FUNCTION_BLOCK Axis EXTENDS CyclicComponent IMPLEMENTS I_Initializable, I_Axis
VAR
	_Axis				 : REFERENCE TO AXIS_REF;
	Defaults			 : ST_MotionDefaults;
	MotionTaskCollection : MotionTaskCollection<ApplicationBaseMotionParameterNc2.MaxMotionTasks>(THIS^);

	// Tasks
	{attribute 'hide'}
	PowerTask : PowerTask := (Name := 'MC Power');
	{attribute 'hide'}
	JogTask : MoveJogTask := (Name := 'MC Jog');
	{attribute 'hide'}
	_StopTask : I_MotionTask := Defaults.DefaultStopTask;
	{attribute 'hide'}
	_ResetTask : I_MotionTask := Defaults.DefaultResetTask;
	{attribute 'hide'}
	_HomeTask : I_MotionTask := Defaults.DefaultHomeTask;

	//
	{attribute 'hide'}
	MCReadParameterSet : MC_ReadParameterSet;
	_AxisParameters	   : ST_AxisParameterSet;
	{attribute 'hide'}
	_Initialized : BOOL;
	{attribute 'hide'}
	_Acceleration : LREAL;
	{attribute 'hide'}
	_Deceleration : LREAL;
	{attribute 'hide'}
	_Velocity : LREAL;
	{attribute 'hide'}
	_Jerk		  : LREAL;
	_McBufferMode : MC_BufferMode;
	_MoveOptions  : ST_MoveOptions;
END_VAR

{attribute 'monitoring' := 'call'}
PROPERTY Acceleration : LREAL
GET
Acceleration := _Acceleration;
END_GET
SET
_Acceleration := Acceleration;
END_SET
END_PROPERTY

{attribute 'monitoring' := 'call'}
PROPERTY ActualAcceleration : LREAL
GET
ActualAcceleration := _Axis.NcToPlc.ActAcc;
END_GET
END_PROPERTY

{attribute 'monitoring' := 'call'}
PROPERTY ActualPosition : LREAL
GET
ActualPosition := _Axis.NcToPlc.ActPos;
END_GET
END_PROPERTY

{attribute 'monitoring' := 'call'}
PROPERTY ActualPositionModulo : LREAL
GET
ActualPositionModulo := _Axis.NcToPlc.ModuloActPos;
END_GET
END_PROPERTY

{attribute 'monitoring' := 'call'}
PROPERTY ActualTorque : LREAL
GET
ActualTorque := _Axis.NcToPlc.ActTorque;
END_GET
END_PROPERTY

{attribute 'monitoring' := 'call'}
PROPERTY ActualVelocity : LREAL
GET
ActualVelocity := _Axis.NcToPlc.ActVelo;
END_GET
END_PROPERTY

PROPERTY Axis : REFERENCE TO AXIS_REF
GET
Axis REF= _Axis;
END_GET
END_PROPERTY

PROPERTY AxisParameterSet : REFERENCE TO ST_AxisParameterSet
GET
AxisParameterSet REF= _AxisParameters;
END_GET
END_PROPERTY

PROPERTY BufferMode : REFERENCE TO MC_BufferMode
GET
BufferMode REF= _McBufferMode;
END_GET
END_PROPERTY

{attribute 'monitoring' := 'call'}
PROPERTY Busy : BOOL
GET
Busy := MotionTaskCollection.Busy;
END_GET
END_PROPERTY

METHOD CyclicLogic
IF NOT _Initialized THEN
	Initialize();
	RETURN;
END_IF

_Axis.ReadStatus();
MotionTaskCollection.CyclicLogic();
END_METHOD

{attribute 'monitoring' := 'call'}
PROPERTY Deceleration : LREAL
GET
Deceleration := _Deceleration;
END_GET
SET
_Deceleration := Deceleration;
END_SET
END_PROPERTY

METHOD Disable
PowerTask.Disable();
END_METHOD

METHOD Enable
IF Error THEN
	RETURN;
END_IF

PowerTask.Enable();
END_METHOD

{attribute 'monitoring' := 'call'}
PROPERTY Enabled : BOOL
GET
Enabled := PowerTask.Enabled;
END_GET
END_PROPERTY

{attribute 'monitoring' := 'call'}
PROPERTY Error : BOOL
GET
Error := MotionTaskCollection.Error OR _Axis.Status.Error;
END_GET
END_PROPERTY

{attribute 'monitoring' := 'call'}
PROPERTY ErrorId : UDINT
GET
IF _Axis.Status.ErrorID <> 0 THEN
	ErrorId := _Axis.Status.ErrorID;
	RETURN;
END_IF

ErrorId := MotionTaskCollection.ErrorId;
END_GET
END_PROPERTY

(*FB_Init is always available implicitly and it is used primarily for initialization.
The return value is not evaluated. For a specific influence, you can also declare the
methods explicitly and provide additional code there with the standard initialization
code. You can evaluate the return value.*)
METHOD FB_Init : BOOL
VAR_INPUT
	(* TRUE: the retain variables are initialized (reset warm / reset cold)*)
	bInitRetains : BOOL;

	(* TRUE: the instance will be copied to the copy code afterward (online change)   *)
	bInCopyCode : BOOL;
	Name		: T_MaxString;
	Axis		: REFERENCE TO AXIS_REF;
END_VAR
_Axis REF= Axis;

// Register all Motion Tasks to Collection
MotionTaskCollection.AddTask(PowerTask);
MotionTaskCollection.AddTask(_StopTask);
MotionTaskCollection.AddTask(_ResetTask);
MotionTaskCollection.AddTask(_HomeTask);
MotionTaskCollection.AddTask(JogTask);
END_METHOD

METHOD Home
VAR_INPUT
END_VAR
_HomeTask.Execute();
END_METHOD

PROPERTY HomeTask : I_MotionTask
SET
MotionTaskCollection.RemoveTaskByInstance(_HomeTask);
_HomeTask := HomeTask;
MotionTaskCollection.AddTask(_HomeTask);
END_SET
END_PROPERTY

{attribute 'monitoring' := 'call'}
PROPERTY InhibitFeedBackward : BOOL
GET
InhibitFeedBackward := PowerTask.InhibitFeedBackward;
END_GET
SET
PowerTask.InhibitFeedBackward := InhibitFeedBackward;
END_SET
END_PROPERTY

{attribute 'monitoring' := 'call'}
PROPERTY InhibitFeedForward : BOOL
GET
InhibitFeedForward := PowerTask.InhibitFeedForward;
END_GET
SET
PowerTask.InhibitFeedForward := InhibitFeedForward;
END_SET
END_PROPERTY

METHOD Initialize
IF NOT _Initialized THEN
	MCReadParameterSet(Parameter := _AxisParameters, Axis := _Axis, Execute := TRUE);
	IF NOT MCReadParameterSet.Busy THEN
		IF MCReadParameterSet.Error THEN
			Trace.LogMessage(_Name, 'Axis not initialized - McReadParameter failed!');
		ELSIF MCReadParameterSet.Done THEN
			_Velocity	  := _AxisParameters.fVeloSlowManual;
			_Acceleration := _AxisParameters.fAcceleration;
			_Deceleration := _AxisParameters.fDeceleration;
			_Jerk		  := _AxisParameters.fJerk;
			Trace.LogMessage(_Name, 'Axis initialization complete');
			_Initialized := TRUE;
		END_IF

		MCReadParameterSet(Parameter := _AxisParameters, Axis := _Axis, Execute := FALSE);
	END_IF
END_IF
END_METHOD

{attribute 'monitoring' := 'call'}
PROPERTY Initialized : BOOL
GET
Initialized := _Initialized;
END_GET
SET
_Initialized := Initialized;
END_SET
END_PROPERTY

{attribute 'monitoring' := 'call'}
PROPERTY Jerk : LREAL
GET
Jerk := _Jerk;
END_GET
SET
_Jerk := Jerk;
END_SET
END_PROPERTY

METHOD Jog
VAR_INPUT
	JogForward	 : BOOL;
	JogBackwards : BOOL;
	JogMode		 : E_JogMode := E_JogMode.MC_JOGMODE_STANDARD_SLOW;
	Position	 : LREAL	 := 0;
END_VAR
IF Error THEN
	RETURN;
END_IF

JogTask.JogBackwards := JogBackwards;
JogTask.JogForward	 := JogForward;
JogTask.Position	 := Position;
JogTask.Mode		 := JogMode;
JogTask.Execute();
END_METHOD

PROPERTY MotionTasks : I_MotionTaskCollection
GET
MotionTasks := MotionTaskCollection;
END_GET
END_PROPERTY

PROPERTY MoveOptions : REFERENCE TO ST_MoveOptions
GET
MoveOptions REF= _MoveOptions;
END_GET
END_PROPERTY

{attribute 'monitoring' := 'call'}
PROPERTY Override : LREAL
SET
PowerTask.Override := Override;
END_SET
END_PROPERTY

{attribute 'monitoring' := 'call'}
PROPERTY PositionLag : LREAL
GET
PositionLag := _Axis.NcToPlc.PosDiff;
END_GET
END_PROPERTY

METHOD RegisterWithParent
VAR_INPUT
	Parent : I_ContainComponents;
END_VAR
SUPER^.RegisterWithParent(Parent);
Parent.RegisterInitialize(THIS^);
END_METHOD

METHOD Reset
IF _ResetTask.Execute() THEN
	MotionTaskCollection.Reset();
END_IF
END_METHOD

PROPERTY ResetTask : I_MotionTask
SET
MotionTaskCollection.RemoveTaskByInstance(_ResetTask);
_ResetTask := ResetTask;
MotionTaskCollection.AddTask(_ResetTask);
END_SET
END_PROPERTY

{attribute 'monitoring' := 'call'}
PROPERTY SetAcceleration : LREAL
GET
SetAcceleration := _Axis.NcToPlc.SetAcc;
END_GET
END_PROPERTY

{attribute 'monitoring' := 'call'}
PROPERTY SetPosition : LREAL
GET
SetPosition := _Axis.NcToPlc.SetPos;
END_GET
END_PROPERTY

{attribute 'monitoring' := 'call'}
PROPERTY SetPositionModulo : LREAL
GET
SetPositionModulo := _Axis.NcToPlc.ModuloSetPos;
END_GET
END_PROPERTY

{attribute 'monitoring' := 'call'}
PROPERTY SetVelocity : LREAL
GET
SetVelocity := _Axis.NcToPlc.SetVelo;
END_GET
END_PROPERTY

METHOD Stop
IF Error AND _Axis.Status.Error THEN
	(* It's possible that a function block errored but
	not the NC itself--in this case we can allow a stop command.
	If the NC Axis has a real fault then we want a successful reset first *)
	RETURN;
END_IF

_StopTask.Execute();
END_METHOD

{attribute 'monitoring' := 'call'}
PROPERTY Stopped : BOOL
GET
Stopped := _Axis.Status.NotMoving;
END_GET
END_PROPERTY

PROPERTY StopTask : I_MotionTask
SET
MotionTaskCollection.RemoveTaskByInstance(_StopTask);
_StopTask := StopTask;
MotionTaskCollection.AddTask(_ResetTask);
END_SET
END_PROPERTY

{attribute 'monitoring' := 'call'}
PROPERTY Velocity : LREAL
GET
Velocity := _Velocity;
END_GET
SET
_Velocity := Velocity;
END_SET
END_PROPERTY

END_FUNCTION_BLOCK

(* stored: Version 1.1.0.1, ProductVersion 3.1.4026.18
   POU Axis: Id {c3c03e8a-759c-4ce9-bcae-63318d943e7c}, SpecialFunc None
   Folder Component: Id {b9674294-e5e8-4857-b2dd-bb9605b4f949}
   Folder Cyclic: Id {cd62d491-a87a-4c24-ab53-621ad021711e}
   Folder Dynamics: Id {393c3e99-a69d-4243-96b4-7490d06ba075}
   Folder Enable: Id {a996dd7a-39c8-423c-9839-645e36a4c7ae}
   Folder Home: Id {e215008b-3961-4321-9331-07c098f36434}
   Folder Initialize: Id {350a9f43-6c08-4c9b-bd16-bb4fcd640dda}
   Folder Jog: Id {b440d357-8c50-41b7-97b2-91a6c011f5d6}
   Folder Reset: Id {853c8cf9-dc4d-4635-94bf-40639ab6791d}
   Folder Status: Id {72a29854-77b1-4e21-8c83-e6fb17183b47}
   Folder Stop: Id {4b02773b-6d51-4517-a15d-46b46992d36e}
   Property Acceleration: Id {bc2c3c5d-a4a9-4cb5-98d3-83a3191a9c81}
   Get Get: Id {6ebbb80e-267f-48b6-bb39-8d2ca4223844}
   Set Set: Id {e0a62beb-1801-4bb4-a76f-99346623f4b9}
   Property ActualAcceleration: Id {b5647fbd-a9d3-4882-8ed1-a0b72765d3b5}
   Get Get: Id {e67bd821-4a1a-44ed-9dc1-bf2f8ef16b0a}
   Property ActualPosition: Id {e1f48912-a935-4b3e-be97-eaceec9cb795}
   Get Get: Id {772eda12-44c2-48fc-8116-a610cf9a6ed0}
   Property ActualPositionModulo: Id {84d10871-a74d-4aa2-a671-8ede5ee35065}
   Get Get: Id {80852d1b-ae4a-43a1-9703-1746633973f5}
   Property ActualTorque: Id {89530b95-2ff6-4521-a671-66d5316590a2}
   Get Get: Id {f1b6f872-58a2-4329-a84d-fe2f48b53e4b}
   Property ActualVelocity: Id {ba440947-68a9-4883-9276-0375868b0a94}
   Get Get: Id {a2f8b812-092f-410b-a402-b7a33bf5b797}
   Property Axis: Id {38c79dbc-ba31-4d4e-8888-4e408cffe3bb}
   Get Get: Id {df4e8fb7-b017-47e2-827b-4155fa44ffd8}
   Property AxisParameterSet: Id {601137f1-5425-4fd4-9a0f-19df82a67e6e}
   Get Get: Id {0e4a2256-1fee-412f-9dac-1fa4f795cf21}
   Property BufferMode: Id {a85af1da-9dee-46aa-bbbb-4758c84e4c91}
   Get Get: Id {d1e71bfd-219f-450d-bb9c-e263de4497af}
   Property Busy: Id {6794a53b-7ced-4307-bcd9-3477d559ac82}
   Get Get: Id {d665c90f-e0eb-4c0b-94cf-47eaad5875d3}
   Method CyclicLogic: Id {10fc0310-6f8d-455a-992b-f31a600e3e01}
   Property Deceleration: Id {db89bb8c-0dcc-4b5f-8969-ffbccd3ee048}
   Get Get: Id {3800a40e-864f-4a8e-a36e-7c389c14756b}
   Set Set: Id {f0482c1d-fb99-4838-a7a8-a7156e0a7edc}
   Method Disable: Id {3bab1b3b-29ff-4bfc-a4eb-0e0f42f5a5b7}
   Method Enable: Id {28103e05-76eb-4b6e-8ca3-aa04ca488039}
   Property Enabled: Id {9c73b2c8-514b-4a7c-998d-28369f5fdf7e}
   Get Get: Id {e85a3e15-6839-4f5c-bb24-c2c90ccdc5cf}
   Property Error: Id {08e691a3-f406-4de1-a788-658111b7a523}
   Get Get: Id {d40a494c-772e-46b9-8af6-4d69798bcac7}
   Property ErrorId: Id {84e4c405-d99b-418e-a3e1-8c72ca915f1b}
   Get Get: Id {ad9aed7a-a7d0-420f-ad7a-1525a3bd7600}
   Method FB_Init: Id {408d8b84-e8bf-4975-a51d-b75b6eec471d}
   Method Home: Id {03b59bd2-3edb-4006-8ed9-515960b2d71c}
   Property HomeTask: Id {853ef4ec-dfa5-43fb-8ffc-aded749a9947}
   Set Set: Id {90777a80-d32c-44e9-9bf9-563776acb7bf}
   Property InhibitFeedBackward: Id {c5c0191f-dbb6-41bc-9c36-d1160afdeefd}
   Get Get: Id {6acb7c40-b74c-4342-8a4f-ca2fab6e2892}
   Set Set: Id {e7024f53-ca04-40e3-a02f-2dfeb6e4123c}
   Property InhibitFeedForward: Id {8959307e-de91-43e2-8d9a-51e4095b0214}
   Get Get: Id {abd49421-29f4-4b77-b708-f285eb3600d1}
   Set Set: Id {1297ae4d-20eb-4797-a6e0-c57453058912}
   Method Initialize: Id {66bade57-0863-4af8-8c50-55eb772839b1}
   Property Initialized: Id {ebd44c64-aad6-4960-8b2f-81d5f43b19d3}
   Get Get: Id {aeebcb0e-1628-4ae8-a555-fcbd0a81bd80}
   Set Set: Id {d711cfec-da17-49cd-b426-000de5c3217f}
   Property Jerk: Id {96ffb255-e0ba-4312-a90f-7dd965cf71b0}
   Get Get: Id {e557ad60-384a-47e9-b9d7-d4f472924031}
   Set Set: Id {d4cca97a-3aef-4baf-b25b-1a7f540a5b6d}
   Method Jog: Id {c855961c-fd72-4b30-bb3c-30f7dfb030f5}
   Property MotionTasks: Id {cf3fa9ca-401c-41ad-a41f-999b7718040b}
   Get Get: Id {af34f3a0-4554-4bf3-84b6-b53c62f02119}
   Property MoveOptions: Id {1da2f2ad-f531-47ad-aa4b-0b0f086322d9}
   Get Get: Id {52746be8-b5c1-425c-8447-3fc4d902eaf9}
   Property Override: Id {c74d8be7-5bb5-4058-b076-f4ab4c78f08d}
   Set Set: Id {6d85d497-c707-42cc-96c7-77ba644e0f08}
   Property PositionLag: Id {f7f4f353-aa5d-44bc-b83d-404ab44f3971}
   Get Get: Id {8d18bf9c-762e-4eb3-abdd-d1b7a4ac6007}
   Method RegisterWithParent: Id {7c253cad-8e86-46be-a1de-97f3fe4d6992}
   Method Reset: Id {4345ab78-8abd-4dc4-8462-07064700c600}
   Property ResetTask: Id {b49f90e4-bf55-4e04-8fe2-be9f3fad9f2b}
   Set Set: Id {fdd59bab-1a03-4da3-9a94-3abd49a82240}
   Property SetAcceleration: Id {9bd86b21-0a70-46d7-952f-db9b168b0ce1}
   Get Get: Id {d7cebf73-953d-4a28-8c6d-d0400f45a387}
   Property SetPosition: Id {5d119d9f-00a0-4eca-a9bd-7cd52817e416}
   Get Get: Id {bab013fd-a2b7-43d7-8d0a-cac9d0832d87}
   Property SetPositionModulo: Id {b3028874-b09c-4bc2-b47a-1f949c20e5ac}
   Get Get: Id {fa858776-d532-4176-9043-6194dab02039}
   Property SetVelocity: Id {3e4ef1ab-63fe-4ccd-aebe-27b7551635ad}
   Get Get: Id {3aa45f93-0793-4119-be6b-a60ae9d4d15f}
   Method Stop: Id {0be87652-03f5-4e18-8106-42910ca0c5b3}
   Property Stopped: Id {766a8887-0006-457a-a31d-6ae62af64552}
   Get Get: Id {6eaf65ce-c6c7-44f6-af26-5e9711f1e1c8}
   Property StopTask: Id {9f0111fe-5c48-4077-a88d-28d745c064e6}
   Set Set: Id {515b1767-8ac6-4ab4-8df1-e6f6fe4b06b0}
   Property Velocity: Id {942585ae-0bea-4380-ad19-28b1e6ed294f}
   Get Get: Id {6ff1ab23-d51f-46cd-9b07-d111af3c7808}
   Set Set: Id {8f7749c3-203e-4b0b-acd3-8f08a5d8d204} *)
